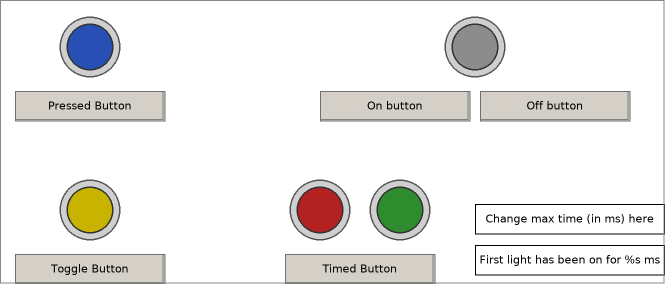
VISUALIZATION Visualization  // 665x284
    Button (15,91 150x30), "Pressed Button"
        tap MAIN.bIsButtonPressed
    Button (15,254 150x30), "Toggle Button", pressed state: main.bIsToggleButtonOn
        tap MAIN.bIsToggleButtonOn
    Button (285,254 150x30), "Timed Button"
        tap main.bIsTimeButtonPressed
    Lamp1 (55,12 70x70), variable: MAIN.fbPressedButton.bLightOfPressedButton, style: Lamp-Lamp1-Blue
    Lamp1 (440,12 70x70), variable: MAIN.fbOnAndOffButtons.bLightOfOnAndOffButton, style: Lamp-Lamp1-Gray
    Lamp1 (55,175 70x70), variable: MAIN.fbToggleButton.bLightOfToggleButton, style: Lamp-Lamp1-Yellow
    Lamp1 (285,175 70x70), variable: MAIN.fbTimedButton.bLightOfTimedButton, style: Lamp-Lamp1-Red
    Lamp1 (365,175 70x70), variable: MAIN.fbTimedButton.bLightOfOtherButton, style: Lamp-Lamp1-Green
    Rectangle (475,245 190x30), "First light has been on for %s ms", text variable: MAIN.fbTimedButton.tTimePressed
    Rectangle (475,204 190x30), "Change max time (in ms) here"
        OnMouseClick: write MAIN.fbTimedButton.sMaxTime via Default
    Button (320,91 150x30), "On button"
        tap MAIN.bIsButtonOn
    Button (480,91 150x30), "Off button"
        tap MAIN.bIsButtonOff
END_VISUALIZATION

(* stored: Version 1.1.0.1, ProductVersion 3.1.4024.12
   Visu Visualization: Id {0ab9e60c-4697-429f-a4ff-cc267fe8084c} *)
